// TIA Portal V20 export
TYPE "LConSMC_typePIDControllerOut"
// stored: Access Published
   STRUCT
      busy : Bool := FALSE;   // TRUE: Der Funktionsbaustein ist aktiv / TRUE: Function block is active
      error : Bool := FALSE;   // TRUE: Es ist ein Fehler aufgetreten / TRUE: An error occured
      errorID : DWord := 16#0000_0000;   // Detaillierte Fehlerbeschreibung / Detailed error description
      upperLimitReached : Bool := FALSE;   // TRUE: Oberer Grenzwert erreicht / TRUE: Upper limit reached
      lowerLimitReached : Bool := FALSE;   // TRUE: Unterer Grenzwert erreicht / TRUE: Lower limit reached
      deviationValue : LReal := 0.0;   // Regelabweichung nach dem Totband / Controller deviation after the deadband filter
      pOutValue : LReal := 0.0;   // P-Komponente des Ausgangs vor der Begrenzung / P component output before limitation
      iOutValue : LReal;   // I-Komponente des Ausgangs vor der Begrenzung / I component output before limitation
      dOutValue : LReal;   // D-Komponente des Ausgangs vor der Begrenzung / D component output before limitation
      outValue : LReal := 0.0;   // Reglerausgang nach Begrenzung und Skalierung / Controller output after limitation and scaling
   END_STRUCT;
END_TYPE
